// TIA Portal V17 export
// export: Created 2025-03-05T08:01:35.5066848Z, ExportSetting WithDefaults, DisplayName Totally Integrated Automation Portal, DisplayVersion V17 Update 8, DisplayName TIA Portal Openness, DisplayVersion V17 Update 8, DisplayName TIA Portal Version Control Interface, DisplayVersion V17, DisplayName SINAMICS Startdrive Advanced, DisplayVersion V17 SP2, DisplayName SINAMICS Startdrive G110M, G120, G120C, G120D, G120P, G115D, DisplayVersion V17 SP2, DisplayName SINAMICS Startdrive G130, G150, S120, S150, SINAMICS MV, S210, DisplayVersion V17 SP2, DisplayName STEP 7 Professional, DisplayVersion V17 Update 8, DisplayName SINUMERIK ONE STEP 7 Toolbox, DisplayVersion V17 Update 12, DisplayName SINUMERIK 840D sl STEP 7 Toolbox, DisplayVersion V17 Update 12, DisplayName STEP 7 Safety, DisplayVersion V17 Update 6, DisplayName WinCC Advanced, DisplayVersion V17 Update 8
FUNCTION "FC10000_GENERAL" : Void   // FC10000, LAD
{ S7_Optimized_Access := 'TRUE' }
VERSION : 0.1
// stored: AutoNumber false, IsIECCheckEnabled false, SetENOAutomatically false, UDAEnableTagReadback false
BEGIN

REGION Network 1: CALL FC10200 PYROMETERS
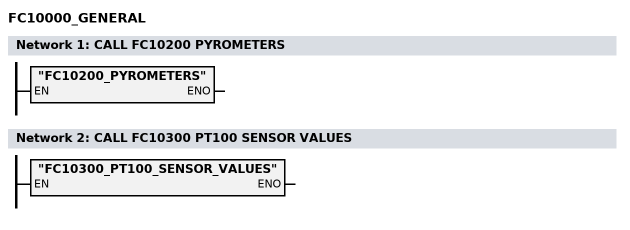
   RUNG wire#powerrail
      "FC10200_PYROMETERS"()
   END_RUNG
   // the same network as SCL:
   "FC10200_PYROMETERS"();
END_REGION

REGION Network 2: CALL FC10300 PT100 SENSOR VALUES
   RUNG wire#powerrail
      "FC10300_PT100_SENSOR_VALUES"()
   END_RUNG
   // the same network as SCL:
   "FC10300_PT100_SENSOR_VALUES"();
END_REGION
END_FUNCTION
